// TIA Portal project "Ryan" (V14)

(* hardware
DEVICE "S71500/ET200MP station_1"  S7-1500 station
   slot 0: "Rail_0"  Rack  6ES7 590-1***0-0AA0
   slot 1: "PLC_1"  CPU 1516-3 PN/DP  6ES7 516-3AN01-0AB0  V2.1
      slot 3: "CPU display_1"  6ES7591-1BA00-0AA0
   slot 2: "DI 32x24VDC HF_1"  DI 32x24VDC HF  6ES7 521-1BL00-0AB0  V2.1
   slot 3: "DQ 32x24VDC/0.5A HF_1"  DQ 32x24VDC/0.5A HF  6ES7 522-1BL01-0AB0  V1.0
   slot 4: "AI 8xU/I/RTD/TC ST_1"  AI 8xU/I/RTD/TC ST  6ES7 531-7KF00-0AB0  V2.1
   slot 5: "AQ 4xU/I ST_1"  AQ 4xU/I ST  6ES7 532-5HD00-0AB0  V2.1
DEVICE "PC station"  SIMATIC PC station
   slot 0: "PC station"  Rail  SIMATIC PC-Station  V1.0
      slot 125: "Stationmanager"  Station_Manager  V6.0.4
   slot 1: "IE general_1"  IE General  IE_CP  V8.2.0
   slot 3: "HMI_RT_1"  WinCC RT Advanced  6AV2 104-0xxxx-xxxx  14.0.1.0
      slot 33792: "Host interface"  Host interface
DEVICE "S71500/ET200MP station_2"  S7-1500 station
   slot 0: "Rail_0"  Rack  6ES7 590-1***0-0AA0
   slot 1: "PLC_2"  Unspecific CPU 1500  6ES7 5XX-XXXXX-XXXX  V2.1
*)

// ===== PLC "PLC_1"  CPU 1516-3 PN/DP =====

VAR_GLOBAL   // PLC tag table "Default tag table"
   "p1" AT %M0.0 : Bool;
   "Clock_Byte" AT %MB1687 : Byte;
   "Clock_10Hz" AT %M1687.0 : Bool;
   "Clock_5Hz" AT %M1687.1 : Bool;
   "Clock_2.5Hz" AT %M1687.2 : Bool;
   "Clock_2Hz" AT %M1687.3 : Bool;
   "Clock_1.25Hz" AT %M1687.4 : Bool;
   "Clock_1Hz" AT %M1687.5 : Bool;
   "Clock_0.625Hz" AT %M1687.6 : Bool;
   "Clock_0.5Hz" AT %M1687.7 : Bool;
   "p2" AT %M0.1 : Bool;
   "p3" AT %M0.2 : Bool;
   "p4" AT %M0.3 : Bool;
   "p5" AT %M0.4 : Bool;
   "p6" AT %M0.5 : Bool;
   "p8" AT %M0.7 : Bool;
   "p9" AT %M1.0 : Bool;
   "p11" AT %M1.2 : Bool;
   "p12" AT %M1.3 : Bool;
   "p13" AT %M1.4 : Bool;
   "p15" AT %M1.6 : Bool;
   "p16" AT %M1.7 : Bool;
   "t1" AT %M2.0 : Bool;
   "t2" AT %M2.1 : Bool;
   "t3" AT %M2.2 : Bool;
   "t4" AT %M2.3 : Bool;
   "t5" AT %M2.4 : Bool;
   "t6" AT %M2.5 : Bool;
   "t7" AT %M2.6 : Bool;
   "t8" AT %M2.7 : Bool;
   "t9" AT %M3.0 : Bool;
   "t10" AT %M3.1 : Bool;
   "t12" AT %M3.3 : Bool;
   "t13" AT %M3.4 : Bool;
   "t14" AT %M3.5 : Bool;
   "t16" AT %M3.7 : Bool;
   "t17" AT %M4.0 : Bool;
   "t18" AT %M4.1 : Bool;
   "t20" AT %M4.3 : Bool;
   "t21" AT %M4.4 : Bool;
   "h" AT %IW4 : Int;
   "B" AT %M4.5 : Bool;
   "p17" AT %M4.6 : Bool;
   "p18" AT %M4.7 : Bool;
   "p19" AT %M5.0 : Bool;
   "p20" AT %M5.1 : Bool;
   "p21" AT %M5.2 : Bool;
   "p22" AT %M5.3 : Bool;
   "p23" AT %M5.4 : Bool;
   "t22" AT %M5.5 : Bool;
   "t23" AT %M5.6 : Bool;
   "t24" AT %M5.7 : Bool;
   "t25" AT %M6.0 : Bool;
   "t26" AT %M6.1 : Bool;
   "t27" AT %M6.2 : Bool;
   "NB1" AT %I0.2 : Bool;
   "NB2" AT %I0.5 : Bool;
   "aux1" AT %M6.3 : Bool;
   "aux2" AT %M6.4 : Bool;
   "aux3" AT %M6.5 : Bool;
   "aux4" AT %M6.6 : Bool;
   "aux5" AT %M6.7 : Bool;
   "aux6" AT %M7.0 : Bool;
   "aux7" AT %M7.1 : Bool;
   "aux8" AT %M7.2 : Bool;
   "aux9" AT %M7.3 : Bool;
   "aux10" AT %M7.4 : Bool;
   "aux11" AT %M7.5 : Bool;
   "aux12" AT %M7.6 : Bool;
   "aux13" AT %M7.7 : Bool;
   "aux14" AT %M8.0 : Bool;
   "aux15" AT %M8.1 : Bool;
   "aux16" AT %M8.2 : Bool;
   "aux17" AT %M8.3 : Bool;
   "aux18" AT %M8.4 : Bool;
   "aux19" AT %M8.5 : Bool;
   "aux20" AT %M8.6 : Bool;
   "aux21" AT %M8.7 : Bool;
   "init" AT %M9.0 : Bool;
   "presenceDiscrete" AT %M9.1 : Bool;
   "AcqAddRead" AT %MW0 : Int;
   "AcqAddStart" AT %MW10 : Int;
   "AcqAddStop" AT %MW12 : Int;
   "AcqAddWrite" AT %MW14 : Int;
   "AcqDateObservation" AT %MW16 : Int;
   "AcqError" AT %M18.0 : Bool;
   "AcqNewValues" AT %M24.0 : Bool;
   "AcqRun" AT %M30.0 : Bool;
   "AcqRunPrevious" AT %M30.1 : Bool;
   "step" AT %MW20 : Int;
   "startTable" AT %MW22 : Int;
   "AcqValues" AT %MD26 : DInt;
   "AcqPrevValues" AT %MD32 : DInt;
   "Timer" AT %T0 : Timer;
   "Time" AT %MD36 : Time;
   "InTime" AT %M0.6 : Bool;
   "TimerOutput" AT %M3.2 : Bool;
   "Done_Signal" AT %M40.0 : Bool;
   "Busy" AT %M40.1 : Bool;
   "Error" AT %M40.2 : Bool;
   "Status" AT %MW42 : Word;
   "Done_Write" AT %M44.0 : Bool;
   "Busy_Write" AT %M44.1 : Bool;
   "Error_Write" AT %M44.2 : Bool;
   "Status_Write" AT %MW46 : Word;
   "Done_Open" AT %M48.0 : Bool;
   "Busy_Open" AT %M48.1 : Bool;
   "Error_Open" AT %M48.2 : Bool;
   "Status_Open" AT %MW50 : Word;
   "id" AT %MD52 : DWord;
   "startAcquisition" AT %M3.6 : Bool;
   "stopAcquisition" AT %M4.2 : Bool;
   "DataLogCreated" AT %M9.2 : Bool;
   "aux22" AT %M9.3 : Bool;
   "createDL" AT %M9.4 : Bool;
   "openDL" AT %M9.5 : Bool;
   "writeDL" AT %M9.6 : Bool;
   "DeleteDL" AT %M9.7 : Bool;
   "closeDL" AT %M18.1 : Bool;
   "p24" AT %M18.2 : Bool;
   "p25" AT %M18.3 : Bool;
   "t28" AT %M18.4 : Bool;
   "t29" AT %M18.5 : Bool;
   "aux23" AT %M18.6 : Bool;
   "mag2count" AT %MW56 : Int;
   "aux24" AT %M18.7 : Bool;
   "Tag_1" AT %T30 : Timer;
   "t30" AT %M19.0 : Bool;
   "Tag_2" AT %T31 : Timer;
   "t31" AT %M19.1 : Bool;
   "p26" AT %M19.2 : Bool;
   "p27" AT %M19.3 : Bool;
   "t32" AT %M19.4 : Bool;
   "resetMag2counter" AT %M19.5 : Bool;
   "aux25" AT %M19.6 : Bool;
END_VAR

VAR_GLOBAL   // PLC tag table "IOVEC"
   "o" AT %I1.6 : Bool;
   "m" AT %I1.7 : Bool;
   "s1" AT %I2.2 : Bool;
   "s2" AT %I2.1 : Bool;
   "s3" AT %I2.0 : Bool;
   "r1" AT %I1.5 : Bool;
   "r2" AT %I1.3 : Bool;
   "r3" AT %I1.1 : Bool;
   "f1" AT %I1.4 : Bool;
   "f2" AT %I1.2 : Bool;
   "f3" AT %I1.0 : Bool;
   "rmag1" AT %I0.1 : Bool;
   "rmag2" AT %I0.4 : Bool;
   "fmag1" AT %I0.0 : Bool;
   "fmag2" AT %I0.3 : Bool;
   "Amag1" AT %Q1.0 : Bool;
   "Amag2" AT %Q1.2 : Bool;
   "Retmag1" AT %Q1.1 : Bool;
   "Retmag2" AT %Q1.3 : Bool;
   "C" AT %Q1.4 : Bool;
   "Pus1" AT %Q0.2 : Bool;
   "Pus2" AT %Q0.1 : Bool;
   "Pus3" AT %Q0.0 : Bool;
END_VAR

DATA_BLOCK "Data_block_1"   // DB1
{ S7_Optimized_Access := 'TRUE' }
VERSION : 0.1
   VAR
      "%I0.0" : Bool;
      "%I0.1" : Bool;
      "%I0.2" : Bool;
      "%I0.3" : Bool;
      "%I0.4" : Bool;
      "%I0.5" : Bool;
      "%I1.0" : Bool;
      "%I1.1" : Bool;
      "%I1.2" : Bool;
      "%I1.3" : Bool;
      "%I1.4" : Bool;
      "%I1.5" : Bool;
      "%I1.6" : Bool;
      "%I1.7" : Bool;
      "%I2.0" : Bool;
      "%I2.1" : Bool;
      "%I2.2" : Bool;
      "%IW4" : Int;
      "%Q0.0" : Bool;
      "%Q0.1" : Bool;
      "%Q0.2" : Bool;
      "%Q1.0" : Bool;
      "%Q1.1" : Bool;
      "%Q1.2" : Bool;
      "%Q1.3" : Bool;
      "%Q1.4" : Bool;
   END_VAR
BEGIN
END_DATA_BLOCK

DATA_BLOCK "DataLog_vars"   // DB3
{ S7_Optimized_Access := 'TRUE' }
VERSION : 0.1
   VAR
      "Name" : String := 'iovectors2';
      ID : DWord := 0;
      Headers : String := 'IOvector';
      Data : Struct
         IOvector : DInt;
      END_STRUCT;
   END_VAR
BEGIN
END_DATA_BLOCK

DATA_BLOCK "DataLog_vars2"   // DB7
{ S7_Optimized_Access := 'TRUE' }
VERSION : 0.1
   VAR
      "Name" : String := 'Test201904081147';
      ID : DWord;
      Header : String := 'Time,IOvector';
      Data : Struct
         "Time" : Time;
         IOvector : DInt;
      END_STRUCT;
   END_VAR
BEGIN
END_DATA_BLOCK

DATA_BLOCK "Runtime"   // DB12
{ S7_Optimized_Access := 'TRUE' }
VERSION : 0.1
   VAR
      ob : OB_Any := 123;
      info : Array[0..4] of LTime;
      retval : Array[0..4] of Int;
   END_VAR
BEGIN
END_DATA_BLOCK

DATA_BLOCK "DATALOGDATA"   // DB16
{ S7_Optimized_Access := 'TRUE' }
VERSION : 0.1
   VAR
      IOVECNAMES : Array[0..22] of String;
      IOVEC : Array[0..22] of Bool;
      AcqValues : Array[0..22] of Bool;
      AcqValuesprev : Array[0..22] of Bool;
      Data : Struct
         o : Bool;
         "m" : Bool;
         s1 : Bool;
         s2 : Bool;
         s3 : Bool;
         r1 : Bool;
         r2 : Bool;
         r3 : Bool;
         f1 : Bool;
         f2 : Bool;
         f3 : Bool;
         rmag1 : Bool;
         rmag2 : Bool;
         fmag1 : Bool;
         fmag2 : Bool;
         Amag1 : Bool;
         Amag2 : Bool;
         Retmag1 : Bool;
         Retmag2 : Bool;
         C : Bool;
         Pus1 : Bool;
         Pus2 : Bool;
         Pus3 : Bool;
      END_STRUCT;
      header : String;
      ID : DWord;
   END_VAR
BEGIN
   IOVECNAMES[1] := 'm';
   IOVECNAMES[2] := 's1';
   IOVECNAMES[3] := 's2';
   IOVECNAMES[4] := 's3';
   IOVECNAMES[5] := 'r1';
   IOVECNAMES[6] := 'r2';
   IOVECNAMES[7] := 'r3';
   IOVECNAMES[8] := 'f1';
   IOVECNAMES[9] := 'f2';
   IOVECNAMES[10] := 'f3';
   IOVECNAMES[11] := 'rmag1';
   IOVECNAMES[12] := 'rmag2';
   IOVECNAMES[13] := 'fmag1';
   IOVECNAMES[14] := 'fmag2';
   IOVECNAMES[15] := 'Amag1';
   IOVECNAMES[16] := 'Amag2';
   IOVECNAMES[17] := 'Retmag1';
   IOVECNAMES[18] := 'Retmag2';
   IOVECNAMES[19] := 'C';
   IOVECNAMES[20] := 'Pus1';
   IOVECNAMES[21] := 'Pus2';
   IOVECNAMES[22] := 'Pus3';
   IOVECNAMES[0] := 'o';
END_DATA_BLOCK

DATA_BLOCK "LOGDATA_DB"   // DB17
{ S7_Optimized_Access := 'TRUE' }
VERSION : 0.1
// stored: InstanceOfName LOGDATA
"LOGDATA"
BEGIN
END_DATA_BLOCK

DATA_BLOCK "DATALOG"   // DB18
{ S7_Optimized_Access := 'TRUE' }
VERSION : 0.1
   VAR
      ACQValues : Array[1..23] of Bool;
   END_VAR
BEGIN
END_DATA_BLOCK

// folder: System blocks/Program resources

DATA_BLOCK "IEC_Timer_0_DB"   // DB6
{ S7_Optimized_Access := 'TRUE' }
AUTHOR : Simatic
FAMILY : IEC
NAME : IEC_TMR
VERSION : 1.0
// stored: InstanceOfName IEC_TIMER
"IEC_TIMER"
BEGIN
END_DATA_BLOCK

DATA_BLOCK "IEC_Timer_0_DB_1"   // DB10
{ S7_Optimized_Access := 'TRUE' }
AUTHOR : Simatic
FAMILY : IEC
NAME : IEC_TMR
VERSION : 1.0
// stored: InstanceOfName IEC_TIMER
"IEC_TIMER"
BEGIN
END_DATA_BLOCK

DATA_BLOCK "IEC_Timer_0_DB_2"   // DB11
{ S7_Optimized_Access := 'TRUE' }
AUTHOR : Simatic
FAMILY : IEC
NAME : IEC_TMR
VERSION : 1.0
// stored: InstanceOfName IEC_TIMER
"IEC_TIMER"
BEGIN
END_DATA_BLOCK

DATA_BLOCK "IEC_Timer_0_DB_3"   // DB13
{ S7_Optimized_Access := 'TRUE' }
AUTHOR : Simatic
FAMILY : IEC
NAME : IEC_TMR
VERSION : 1.0
// stored: InstanceOfName IEC_TIMER
"IEC_TIMER"
BEGIN
END_DATA_BLOCK

DATA_BLOCK "IEC_Timer_0_DB_4"   // DB14
{ S7_Optimized_Access := 'TRUE' }
AUTHOR : Simatic
FAMILY : IEC
NAME : IEC_TMR
VERSION : 1.0
// stored: InstanceOfName IEC_TIMER
"IEC_TIMER"
BEGIN
END_DATA_BLOCK

DATA_BLOCK "IEC_Counter_0_DB"   // DB15
{ S7_Optimized_Access := 'TRUE' }
AUTHOR : Simatic
FAMILY : IEC
NAME : CNTR
VERSION : 1.0
// stored: InstanceOfName IEC_COUNTER
"IEC_COUNTER"
BEGIN
END_DATA_BLOCK

// folder: (top level)

ORGANIZATION_BLOCK "Main"   // OB1, LAD, ProgramCycle
TITLE = "Main Program Sweep (Cycle)"
{ S7_Optimized_Access := 'FALSE' }
VERSION : 0.1
   VAR_TEMP
      EV_CLASS : Byte;   // Bits 0-3 = 1:Coming event, Bits 4-7 = 1:Event class 1
      SCAN_1 : Byte;   // 1:Initial call of the OB, 3: Call 2-n of the OB
      PRIORITY : Byte;   // Priority of OB Execution
      OB_NUMBR : Byte;   // OB number
      RESERVED_1 : Byte;   // Reserved for system
      RESERVED_2 : Byte;   // Reserved for system
      PREV_CYCLE : Int;   // Previous program cycle time (milliseconds)
      MIN_CYCLE : Int;   // Minimum program cycle time (milliseconds)
      MAX_CYCLE : Int;   // Maximum program cycle time (milliseconds)
      DATE_TIME : Date_And_Time;   // Date and time OB started
      activateCreate : Bool;
      DataLogAlreadyExists : Bool;
      DeleteDataLog : Bool;
   END_VAR
BEGIN

REGION Network 1
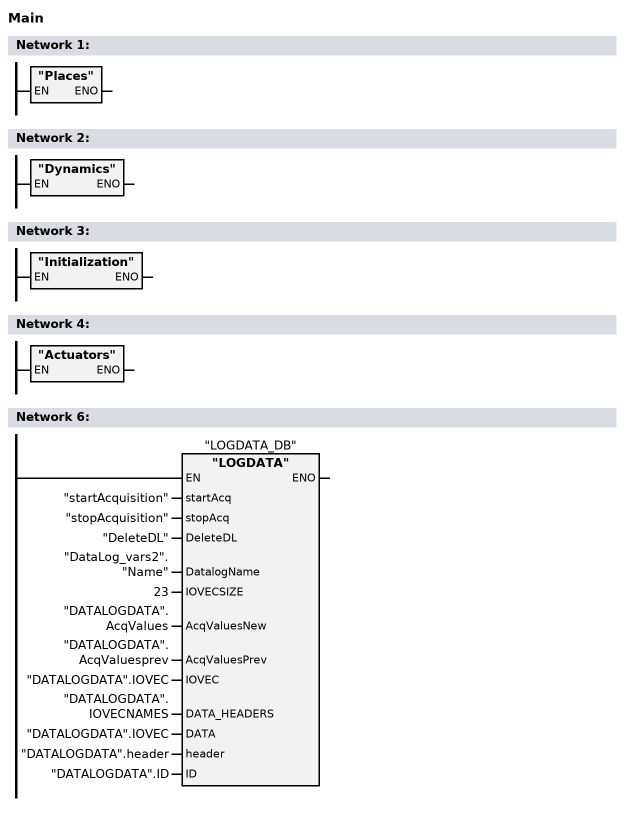
   RUNG wire#powerrail
      "Places"()
   END_RUNG
   // the same network as SCL:
   "Places"();
END_REGION

REGION Network 2
   RUNG wire#powerrail
      "Dynamics"()
   END_RUNG
   // the same network as SCL:
   "Dynamics"();
END_REGION

REGION Network 3
   RUNG wire#powerrail
      "Initialization"()
   END_RUNG
   // the same network as SCL:
   "Initialization"();
END_REGION

REGION Network 4
   RUNG wire#powerrail
      "Actuators"()
   END_RUNG
   // the same network as SCL:
   "Actuators"();
END_REGION

REGION Network 6
   RUNG wire#powerrail
      "LOGDATA_DB"(startAcq := "startAcquisition", stopAcq := "stopAcquisition", DeleteDL := "DeleteDL", DatalogName := "DataLog_vars2"."Name", IOVECSIZE := 23, AcqValuesNew := "DATALOGDATA".AcqValues, AcqValuesPrev := "DATALOGDATA".AcqValuesprev, IOVEC := "DATALOGDATA".IOVEC, DATA_HEADERS := "DATALOGDATA".IOVECNAMES, DATA := "DATALOGDATA".IOVEC, header := "DATALOGDATA".header, ID := "DATALOGDATA".ID)
   END_RUNG
   // the same network as SCL:
   "LOGDATA_DB"(startAcq := "startAcquisition",   // "LOGDATA"
                stopAcq := "stopAcquisition",
                DeleteDL := "DeleteDL",
                DatalogName := "DataLog_vars2"."Name",
                IOVECSIZE := 23,
                AcqValuesNew := "DATALOGDATA".AcqValues,
                AcqValuesPrev := "DATALOGDATA".AcqValuesprev,
                IOVEC := "DATALOGDATA".IOVEC,
                DATA_HEADERS := "DATALOGDATA".IOVECNAMES,
                DATA := "DATALOGDATA".IOVEC,
                header := "DATALOGDATA".header,
                ID := "DATALOGDATA".ID);
END_REGION
END_ORGANIZATION_BLOCK

// folder: LOGGING

FUNCTION_BLOCK "LOGDATA"   // FB1, LAD
{ S7_Optimized_Access := 'TRUE' }
VERSION : 0.1
   VAR_INPUT
      startAcq : Bool;
      stopAcq : Bool;
      DeleteDL : Bool;
      DatalogName : String;
      IOVECSIZE : UDInt;
   END_VAR
   VAR_IN_OUT
      AcqValuesNew : Array[*] of Bool;
      AcqValuesPrev : Array[*] of Bool;
      IOVEC : Array[*] of Bool;
      DATA_HEADERS : Array[*] of String;
      DATA : Variant;
      header : String;
      ID : DWord;
   END_VAR
   VAR_TEMP
      DeleteDatalog : Bool;
      moveBlkVariantRetVal : Int;
      i : Int;
      dataheaderslowerbound : DInt;
      dataheadersupperbound : DInt;
   END_VAR
   VAR_TEMP   // added for the SCL form of the ladder/FBD networks
      _w1 : Bool;
      _w2 : Bool;
   END_VAR
BEGIN

REGION Network 1 (SCL): Name header
       #header := '';
   #dataheaderslowerbound := LOWER_BOUND(ARR := #DATA_HEADERS, DIM := 1);
   #dataheadersupperbound := UPPER_BOUND(ARR := #DATA_HEADERS, DIM := 1);

   FOR #i := #dataheaderslowerbound TO #dataheadersupperbound-1 DO
       // Statement section FOR

       #header := CONCAT(IN1 := #header, IN2 := #DATA_HEADERS[#i]);
       #header := CONCAT(IN1 := #header, IN2 := ',');
   END_FOR;
   #header := CONCAT(IN1 := #header, IN2 := #DATA_HEADERS[#dataheadersupperbound]);
END_REGION

REGION Network 2: Start or stop acquisition
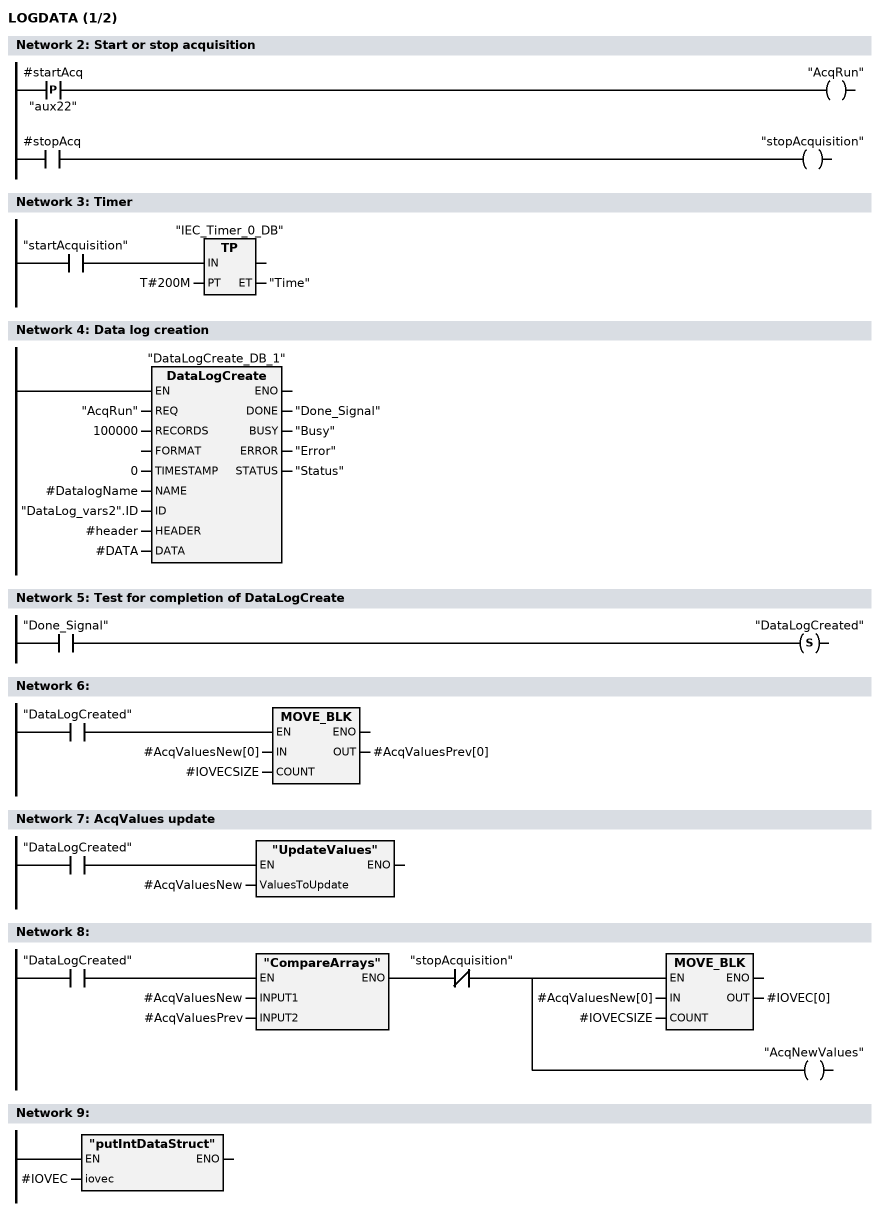
   RUNG wire#powerrail
      P_Contact(operand := #startAcq, bit := "aux22")
      Coil( "AcqRun" )
   END_RUNG
   RUNG wire#powerrail
      Contact( #stopAcq )
      Coil( "stopAcquisition" )
   END_RUNG
   // the same network as SCL:
   #_w1 := #startAcq AND NOT "aux22";   // rising edge of #startAcq
   "aux22" := #startAcq;
   "AcqRun" := #_w1;
   "stopAcquisition" := #stopAcq;
END_REGION

REGION Network 3: Timer
   "IEC_Timer_0_DB".TP(IN := "startAcquisition", PT := T#200M, ET => "Time");
END_REGION

REGION Network 4: Data log creation
   "DataLogCreate_DB_1"(REQ := "AcqRun",   // DataLogCreate
                        RECORDS := 100000,
                        TIMESTAMP := 0,
                        "NAME" := #DatalogName,
                        ID := "DataLog_vars2".ID,
                        HEADER := #header,
                        DATA := #DATA,
                        DONE => "Done_Signal",
                        BUSY => "Busy",
                        ERROR => "Error",
                        STATUS => "Status");
END_REGION

REGION Network 5: Test for completion of DataLogCreate
   RUNG wire#powerrail
      Contact( "Done_Signal" )
      S_Coil( "DataLogCreated" )
   END_RUNG
   // the same network as SCL:
   IF "Done_Signal" THEN "DataLogCreated" := TRUE; END_IF;
END_REGION

REGION Network 6
   IF "DataLogCreated" THEN
       MOVE_BLK(IN := #AcqValuesNew[0], COUNT := #IOVECSIZE, OUT => #AcqValuesPrev[0]);
   END_IF;
END_REGION

REGION Network 7: AcqValues update
   RUNG wire#powerrail
      Contact( "DataLogCreated" )
      "UpdateValues"(ValuesToUpdate := #AcqValuesNew)
   END_RUNG
   // the same network as SCL:
   IF "DataLogCreated" THEN "UpdateValues"(ValuesToUpdate := #AcqValuesNew); END_IF;
END_REGION

REGION Network 8
   "CompareArrays"(EN := "DataLogCreated", INPUT1 := #AcqValuesNew, INPUT2 := #AcqValuesPrev, ENO => #_w1);
   #_w2 := #_w1 AND NOT "stopAcquisition";
   IF #_w2 THEN MOVE_BLK(IN := #AcqValuesNew[0], COUNT := #IOVECSIZE, OUT => #IOVEC[0]); END_IF;
   "AcqNewValues" := #_w2;
END_REGION

REGION Network 9
   RUNG wire#powerrail
      "putIntDataStruct"(iovec := #IOVEC)
   END_RUNG
   // the same network as SCL:
   "putIntDataStruct"(iovec := #IOVEC);
END_REGION

REGION Network 10: Write to data log
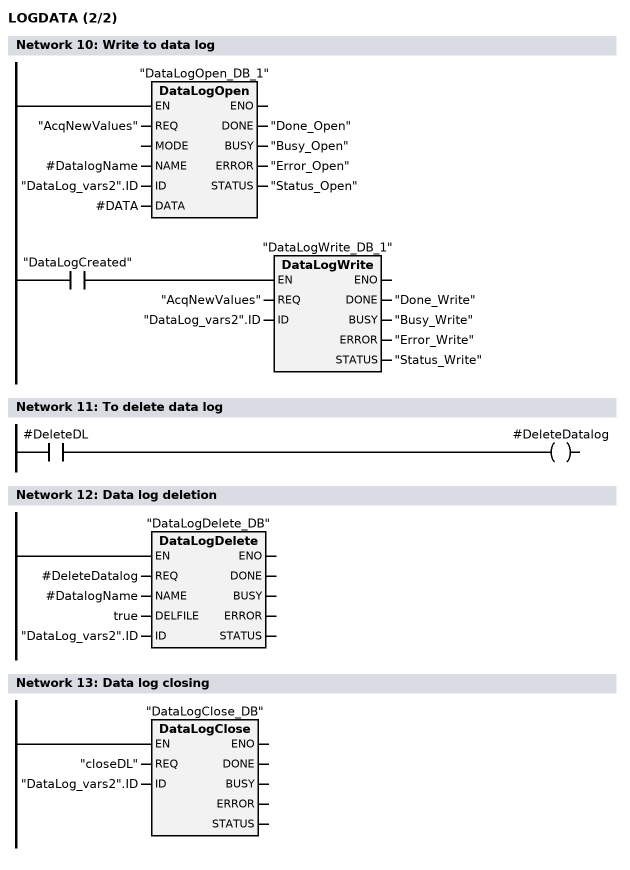
   "DataLogOpen_DB_1"(REQ := "AcqNewValues",   // DataLogOpen
                      "NAME" := #DatalogName,
                      ID := "DataLog_vars2".ID,
                      Data := #DATA,
                      DONE => "Done_Open",
                      BUSY => "Busy_Open",
                      ERROR => "Error_Open",
                      STATUS => "Status_Open");
   IF "DataLogCreated" THEN
       "DataLogWrite_DB_1"(REQ := "AcqNewValues",   // DataLogWrite
                           ID := "DataLog_vars2".ID,
                           DONE => "Done_Write",
                           BUSY => "Busy_Write",
                           ERROR => "Error_Write",
                           STATUS => "Status_Write");
   END_IF;
END_REGION

REGION Network 11: To delete data log
   RUNG wire#powerrail
      Contact( #DeleteDL )
      Coil( #DeleteDatalog )
   END_RUNG
   // the same network as SCL:
   #DeleteDatalog := #DeleteDL;
END_REGION

REGION Network 12: Data log deletion
   "DataLogDelete_DB"(REQ := #DeleteDatalog, "NAME" := #DatalogName, DelFile := true, ID := "DataLog_vars2".ID);   // DataLogDelete
END_REGION

REGION Network 13: Data log closing
   "DataLogClose_DB"(REQ := "closeDL", ID := "DataLog_vars2".ID);   // DataLogClose
END_REGION
END_FUNCTION_BLOCK

FUNCTION "DataLogging" : Void   // FC5, LAD
{ S7_Optimized_Access := 'TRUE' }
VERSION : 0.1
   VAR_INPUT
      startAcq : Bool;
      stopAcq : Bool;
      DeleteDL : Bool;
      DatalogName : String;
   END_VAR
   VAR_TEMP
      DeleteDatalog : Bool;
   END_VAR
   VAR_TEMP   // added for the SCL form of the ladder/FBD networks
      _w1 : Bool;
   END_VAR
BEGIN

REGION Network 1: Start or stop acquisition
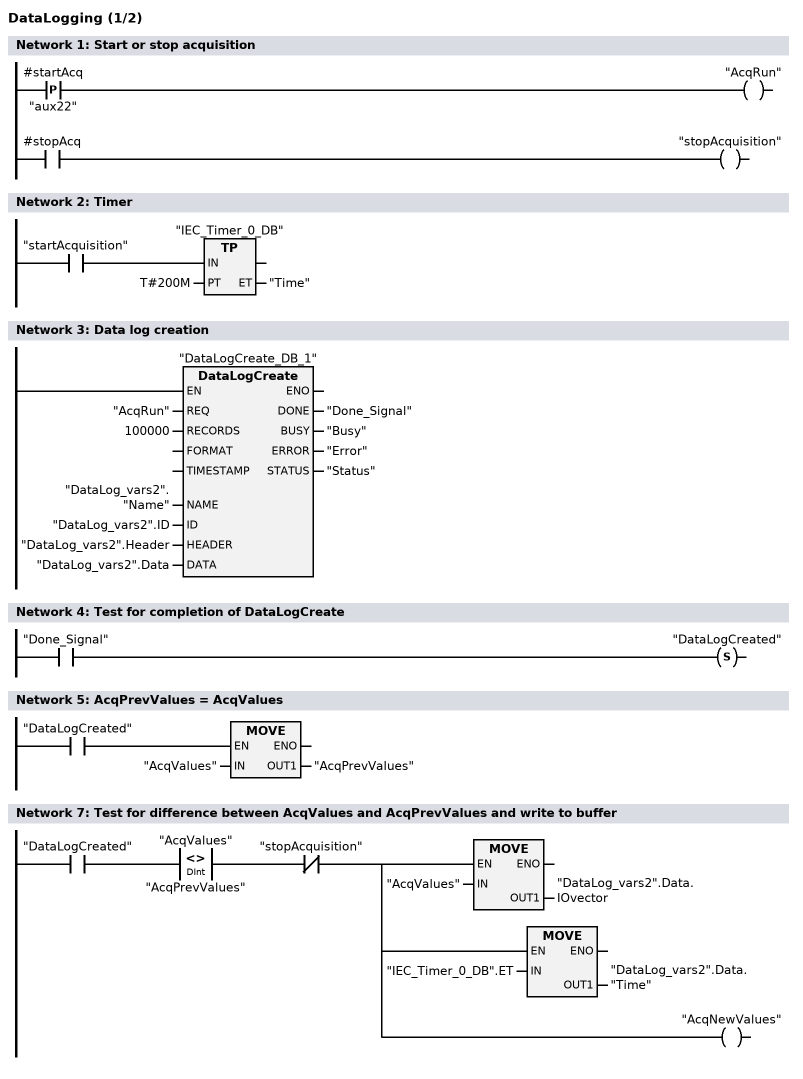
   RUNG wire#powerrail
      P_Contact(operand := #startAcq, bit := "aux22")
      Coil( "AcqRun" )
   END_RUNG
   RUNG wire#powerrail
      Contact( #stopAcq )
      Coil( "stopAcquisition" )
   END_RUNG
   // the same network as SCL:
   #_w1 := #startAcq AND NOT "aux22";   // rising edge of #startAcq
   "aux22" := #startAcq;
   "AcqRun" := #_w1;
   "stopAcquisition" := #stopAcq;
END_REGION

REGION Network 2: Timer
   "IEC_Timer_0_DB".TP(IN := "startAcquisition", PT := T#200M, ET => "Time");
END_REGION

REGION Network 3: Data log creation
   "DataLogCreate_DB_1"(REQ := "AcqRun",   // DataLogCreate
                        RECORDS := 100000,
                        "NAME" := "DataLog_vars2"."Name",
                        ID := "DataLog_vars2".ID,
                        HEADER := "DataLog_vars2".Header,
                        DATA := "DataLog_vars2".Data,
                        DONE => "Done_Signal",
                        BUSY => "Busy",
                        ERROR => "Error",
                        STATUS => "Status");
END_REGION

REGION Network 4: Test for completion of DataLogCreate
   RUNG wire#powerrail
      Contact( "Done_Signal" )
      S_Coil( "DataLogCreated" )
   END_RUNG
   // the same network as SCL:
   IF "Done_Signal" THEN "DataLogCreated" := TRUE; END_IF;
END_REGION

REGION Network 5: AcqPrevValues = AcqValues
   RUNG wire#powerrail
      Contact( "DataLogCreated" )
      Move(in := "AcqValues", out1 => "AcqPrevValues")
   END_RUNG
   // the same network as SCL:
   IF "DataLogCreated" THEN "AcqPrevValues" := "AcqValues"; END_IF;
END_REGION

REGION Network 6 (SCL): AcqValues update
   IF "DataLogCreated" THEN
       "AcqValues".%X0 := "fmag1";
       "AcqValues".%X1 := "rmag1";
       "AcqValues".%X2 := "fmag2";
       "AcqValues".%X3 := "rmag2";
       "AcqValues".%X4 := "f3";
       "AcqValues".%X5 := "r3";
       "AcqValues".%X6 := "f2";
       "AcqValues".%X7 := "r2";
       "AcqValues".%X8 := "f1";
       "AcqValues".%X9 := "r1";
       "AcqValues".%X10 := "o";
       "AcqValues".%X11 := "m";
       "AcqValues".%X12 := "s3";
       "AcqValues".%X13 := "s2";
       "AcqValues".%X14 := "s1";
       "AcqValues".%X15 := "Pus3";
       "AcqValues".%X16 := "Pus2";
       "AcqValues".%X17 := "Pus1";
       "AcqValues".%X18 := "Amag1";
       "AcqValues".%X19 := "Retmag1";
       "AcqValues".%X20 := "Amag2";
       "AcqValues".%X21 := "Retmag2";
       "AcqValues".%X22 := "C";
   END_IF;
END_REGION

REGION Network 7: Test for difference between AcqValues and AcqPrevValues and write to buffer
   RUNG wire#powerrail
      Contact( "DataLogCreated" )
      { S7_Templates := "SrcType := DInt" } NE_Contact(in1 := "AcqValues", in2 := "AcqPrevValues")
      I_Contact( "stopAcquisition" )
      wire#w1
      Move(in := "AcqValues", out1 => "DataLog_vars2".Data.IOvector)
   END_RUNG
   RUNG wire#w1
      Move(in := "IEC_Timer_0_DB".ET, out1 => "DataLog_vars2".Data."Time")
   END_RUNG
   RUNG wire#w1
      Coil( "AcqNewValues" )
   END_RUNG
   // the same network as SCL:
   #_w1 := "DataLogCreated" AND ("AcqValues" <> "AcqPrevValues") AND NOT "stopAcquisition";
   IF #_w1 THEN
       "DataLog_vars2".Data.IOvector := "AcqValues";
       "DataLog_vars2".Data."Time" := "IEC_Timer_0_DB".ET;
   END_IF;
   "AcqNewValues" := #_w1;
END_REGION

REGION Network 8: Write to data log
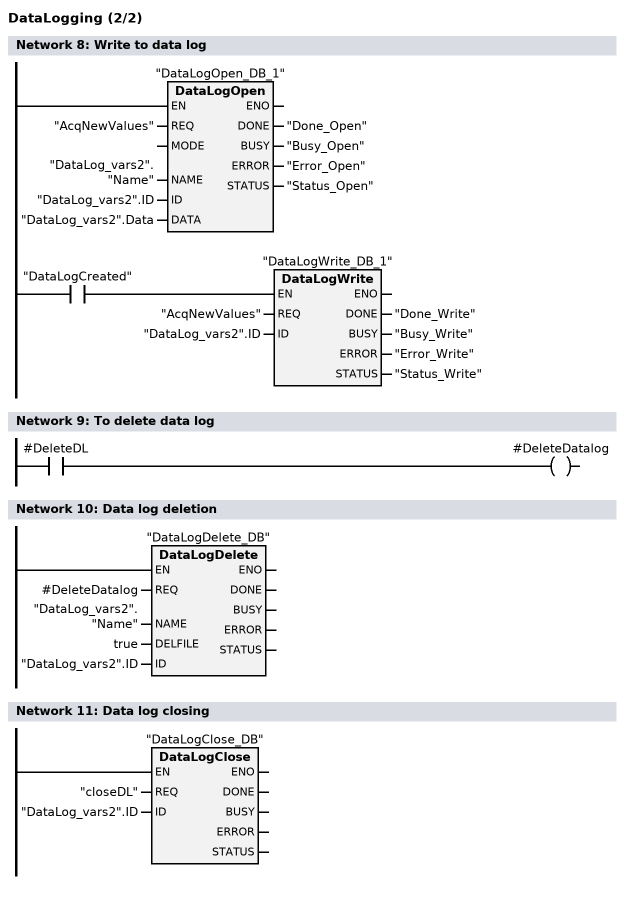
   "DataLogOpen_DB_1"(REQ := "AcqNewValues",   // DataLogOpen
                      "NAME" := "DataLog_vars2"."Name",
                      ID := "DataLog_vars2".ID,
                      Data := "DataLog_vars2".Data,
                      DONE => "Done_Open",
                      BUSY => "Busy_Open",
                      ERROR => "Error_Open",
                      STATUS => "Status_Open");
   IF "DataLogCreated" THEN
       "DataLogWrite_DB_1"(REQ := "AcqNewValues",   // DataLogWrite
                           ID := "DataLog_vars2".ID,
                           DONE => "Done_Write",
                           BUSY => "Busy_Write",
                           ERROR => "Error_Write",
                           STATUS => "Status_Write");
   END_IF;
END_REGION

REGION Network 9: To delete data log
   RUNG wire#powerrail
      Contact( #DeleteDL )
      Coil( #DeleteDatalog )
   END_RUNG
   // the same network as SCL:
   #DeleteDatalog := #DeleteDL;
END_REGION

REGION Network 10: Data log deletion
   "DataLogDelete_DB"(REQ := #DeleteDatalog,   // DataLogDelete
                      "NAME" := "DataLog_vars2"."Name",
                      DelFile := true,
                      ID := "DataLog_vars2".ID);
END_REGION

REGION Network 11: Data log closing
   "DataLogClose_DB"(REQ := "closeDL", ID := "DataLog_vars2".ID);   // DataLogClose
END_REGION

REGION Network 12 (SCL)
   "Runtime".ob := "OB_Main";

   "Runtime".retval[1] := RT_INFO(MODE := 1,
                                  OB := "Runtime".ob,
                                  INFO := "Runtime".info[1]);

   "Runtime".retval[2] := RT_INFO(MODE := 2,
                                  OB := "Runtime".ob,
                                  INFO := "Runtime".info[2]);

   "Runtime".retval[3] := RT_INFO(MODE := 3,
                                  OB := "Runtime".ob,
                                  INFO := "Runtime".info[3]);

   "Runtime".retval[4] := RT_INFO(MODE := 25,
                                  OB := "Runtime".ob,
                                  INFO := "Runtime".info[4]);
END_REGION
END_FUNCTION

FUNCTION "UpdateValues" : Void   // FC6, LAD
{ S7_Optimized_Access := 'TRUE' }
VERSION : 0.1
   VAR_IN_OUT
      ValuesToUpdate : Array[*] of Bool;
   END_VAR
BEGIN

REGION Network 1 (SCL)
   #ValuesToUpdate[0] := "o";
   #ValuesToUpdate[1] := "m";
   #ValuesToUpdate[2] := "s1";
   #ValuesToUpdate[3] := "s2";
   #ValuesToUpdate[4] := "s3";
   #ValuesToUpdate[5] := "r1";
   #ValuesToUpdate[6] := "r2";
   #ValuesToUpdate[7] := "r3";
   #ValuesToUpdate[8] := "f1";
   #ValuesToUpdate[9] := "f2";
   #ValuesToUpdate[10] := "f3";
   #ValuesToUpdate[11] := "rmag1";
   #ValuesToUpdate[12] := "rmag2";
   #ValuesToUpdate[13] := "fmag1";
   #ValuesToUpdate[14] := "fmag2";
   #ValuesToUpdate[15] := "Amag1";
   #ValuesToUpdate[16] := "Amag2";
   #ValuesToUpdate[17] := "Retmag1";
   #ValuesToUpdate[18] := "Retmag2";
   #ValuesToUpdate[19] := "C";
   #ValuesToUpdate[20] := "Pus1";
   #ValuesToUpdate[21] := "Pus2";
   #ValuesToUpdate[22] := "Pus3";
END_REGION
END_FUNCTION

FUNCTION "putIntDataStruct" : Void   // FC8, LAD
{ S7_Optimized_Access := 'TRUE' }
VERSION : 0.1
   VAR_IN_OUT
      iovec : Array[*] of Bool;
   END_VAR
BEGIN

REGION Network 1 (SCL)
   "DATALOGDATA".Data.o := #iovec[0];
   "DATALOGDATA".Data."m" := #iovec[1];
   "DATALOGDATA".Data.s1 := #iovec[2];
   "DATALOGDATA".Data.s2 := #iovec[3];
   "DATALOGDATA".Data.s3 := #iovec[4];
   "DATALOGDATA".Data.r1 := #iovec[5];
   "DATALOGDATA".Data.r2 := #iovec[6];
   "DATALOGDATA".Data.r3 := #iovec[7];
   "DATALOGDATA".Data.f1 := #iovec[8];
   "DATALOGDATA".Data.f2 := #iovec[9];
   "DATALOGDATA".Data.f3 := #iovec[10];
   "DATALOGDATA".Data.rmag1 := #iovec[11];
   "DATALOGDATA".Data.rmag2 := #iovec[12];
   "DATALOGDATA".Data.fmag1 := #iovec[13];
   "DATALOGDATA".Data.fmag2 := #iovec[14];
   "DATALOGDATA".Data.Amag1 := #iovec[15];
   "DATALOGDATA".Data.Amag2 := #iovec[16];
   "DATALOGDATA".Data.Retmag1 := #iovec[17];
   "DATALOGDATA".Data.Retmag2 := #iovec[18];
   "DATALOGDATA".Data.C := #iovec[19];
   "DATALOGDATA".Data.Pus1 := #iovec[20];
   "DATALOGDATA".Data.Pus2 := #iovec[21];
   "DATALOGDATA".Data.Pus3 := #iovec[22];
END_REGION
END_FUNCTION

// folder: LOGGING/utils

FUNCTION "CompareArrays" : Void   // FC7, LAD
{ S7_Optimized_Access := 'TRUE' }
VERSION : 0.1
   VAR_INPUT
      INPUT1 : Array[*] of Bool;
      INPUT2 : Array[*] of Bool;
   END_VAR
   VAR_TEMP
      out : Bool;
      i : Int;
      dataheaderslowerbound : DInt;
      dataheadersupperbound : DInt;
   END_VAR
BEGIN

REGION Network 1 (SCL)
   #out := TRUE;

   #dataheaderslowerbound := LOWER_BOUND(ARR := #INPUT1, DIM := 1);
   #dataheadersupperbound := UPPER_BOUND(ARR := #INPUT1, DIM := 1);

   FOR #i := #dataheaderslowerbound TO #dataheadersupperbound DO
       // Statement section FOR
       #out := #out AND (#INPUT1[#i] = #INPUT2[#i]);

   END_FOR;

   ENO := NOT #out;
END_REGION
END_FUNCTION

// folder: PetriNet

FUNCTION "Places" : Void   // FC1, LAD
{ S7_Optimized_Access := 'TRUE' }
VERSION : 0.1
   VAR_TEMP   // added for the SCL form of the ladder/FBD networks
      _w1 : Bool;
      _w2 : Bool;
      _w3 : Bool;
      _w4 : Bool;
      _w5 : Bool;
      _w6 : Bool;
      _w7 : Bool;
      _w8 : Bool;
      _w9 : Bool;
      _w10 : Bool;
      _w11 : Bool;
      _w12 : Bool;
      _w13 : Bool;
      _w14 : Bool;
      _w15 : Bool;
      _w16 : Bool;
      _w17 : Bool;
      _w18 : Bool;
   END_VAR
BEGIN

REGION Network 1
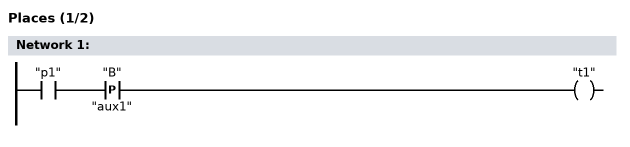
   RUNG wire#powerrail
      Contact( "p1" )
      P_Contact(operand := "B", bit := "aux1")
      Coil( "t1" )
   END_RUNG
   // the same network as SCL:
   #_w1 := "p1" AND "B" AND NOT "aux1";   // rising edge of "B"
   "aux1" := "B";
   "t1" := #_w1;
END_REGION

REGION Network 2: Places
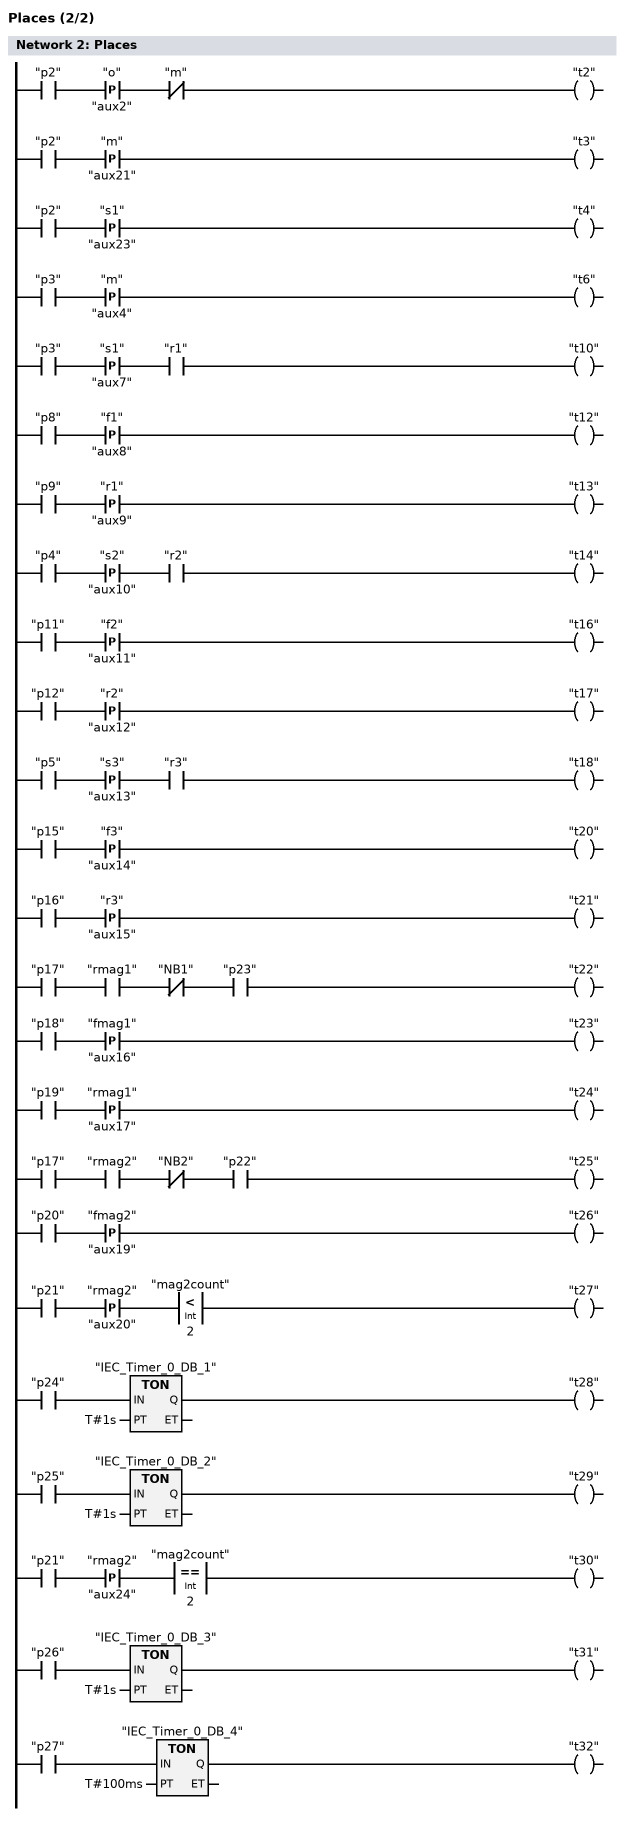
   #_w1 := "p2" AND "o" AND NOT "aux2";   // rising edge of "o"
   "aux2" := "o";
   "t2" := #_w1 AND NOT "m";
   #_w2 := "p2" AND "m" AND NOT "aux21";   // rising edge of "m"
   "aux21" := "m";
   "t3" := #_w2;
   #_w3 := "p2" AND "s1" AND NOT "aux23";   // rising edge of "s1"
   "aux23" := "s1";
   "t4" := #_w3;
   #_w4 := "p3" AND "m" AND NOT "aux4";   // rising edge of "m"
   "aux4" := "m";
   "t6" := #_w4;
   #_w5 := "p3" AND "s1" AND NOT "aux7";   // rising edge of "s1"
   "aux7" := "s1";
   "t10" := #_w5 AND "r1";
   #_w6 := "p8" AND "f1" AND NOT "aux8";   // rising edge of "f1"
   "aux8" := "f1";
   "t12" := #_w6;
   #_w7 := "p9" AND "r1" AND NOT "aux9";   // rising edge of "r1"
   "aux9" := "r1";
   "t13" := #_w7;
   #_w8 := "p4" AND "s2" AND NOT "aux10";   // rising edge of "s2"
   "aux10" := "s2";
   "t14" := #_w8 AND "r2";
   #_w9 := "p11" AND "f2" AND NOT "aux11";   // rising edge of "f2"
   "aux11" := "f2";
   "t16" := #_w9;
   #_w10 := "p12" AND "r2" AND NOT "aux12";   // rising edge of "r2"
   "aux12" := "r2";
   "t17" := #_w10;
   #_w11 := "p5" AND "s3" AND NOT "aux13";   // rising edge of "s3"
   "aux13" := "s3";
   "t18" := #_w11 AND "r3";
   #_w12 := "p15" AND "f3" AND NOT "aux14";   // rising edge of "f3"
   "aux14" := "f3";
   "t20" := #_w12;
   #_w13 := "p16" AND "r3" AND NOT "aux15";   // rising edge of "r3"
   "aux15" := "r3";
   "t21" := #_w13;
   "t22" := "p17" AND "rmag1" AND NOT "NB1" AND "p23";
   #_w14 := "p18" AND "fmag1" AND NOT "aux16";   // rising edge of "fmag1"
   "aux16" := "fmag1";
   "t23" := #_w14;
   #_w15 := "p19" AND "rmag1" AND NOT "aux17";   // rising edge of "rmag1"
   "aux17" := "rmag1";
   "t24" := #_w15;
   "t25" := "p17" AND "rmag2" AND NOT "NB2" AND "p22";
   #_w16 := "p20" AND "fmag2" AND NOT "aux19";   // rising edge of "fmag2"
   "aux19" := "fmag2";
   "t26" := #_w16;
   #_w17 := "p21" AND "rmag2" AND NOT "aux20";   // rising edge of "rmag2"
   "aux20" := "rmag2";
   "t27" := #_w17 AND ("mag2count" < 2);
   "IEC_Timer_0_DB_1".TON(IN := "p24", PT := T#1s);
   "t28" := "IEC_Timer_0_DB_1".Q;
   "IEC_Timer_0_DB_2".TON(IN := "p25", PT := T#1s);
   "t29" := "IEC_Timer_0_DB_2".Q;
   #_w18 := "p21" AND "rmag2" AND NOT "aux24";   // rising edge of "rmag2"
   "aux24" := "rmag2";
   "t30" := #_w18 AND ("mag2count" = 2);
   "IEC_Timer_0_DB_3".TON(IN := "p26", PT := T#1s);
   "t31" := "IEC_Timer_0_DB_3".Q;
   "IEC_Timer_0_DB_4".TON(IN := "p27", PT := T#100ms);
   "t32" := "IEC_Timer_0_DB_4".Q;
END_REGION
END_FUNCTION

FUNCTION "Dynamics" : Void   // FC2, LAD
{ S7_Optimized_Access := 'TRUE' }
VERSION : 0.1
BEGIN

REGION Network 1: Dynamics
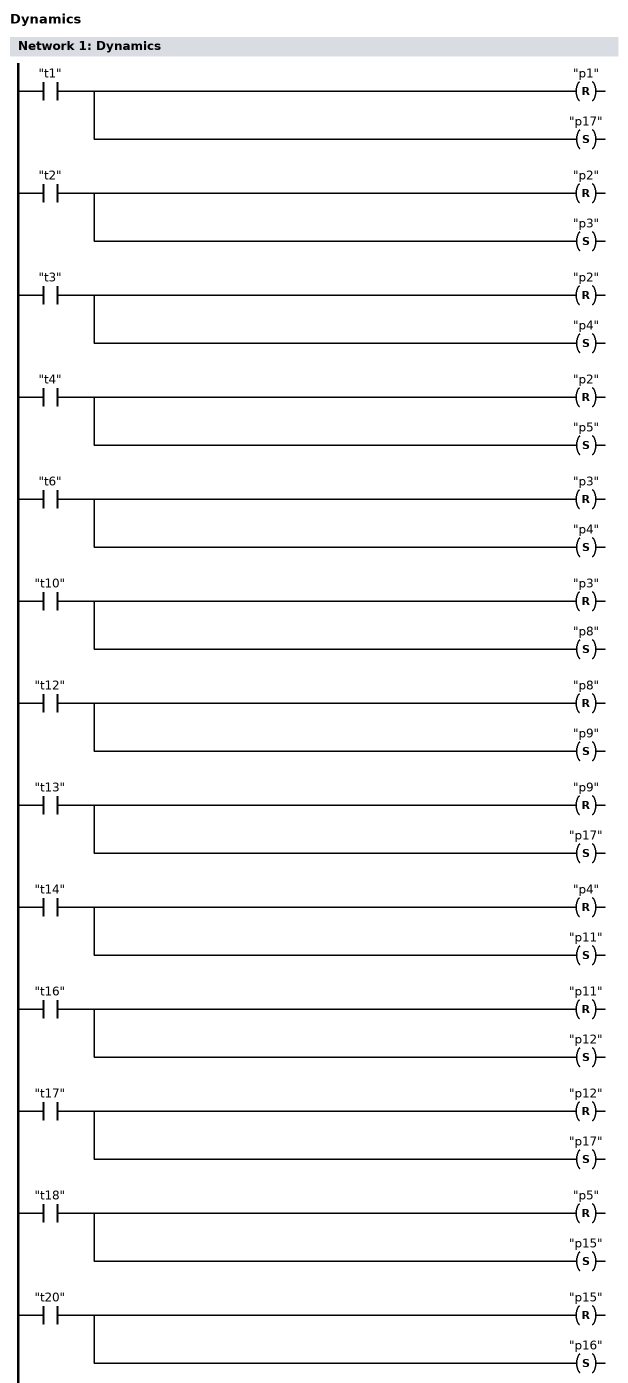
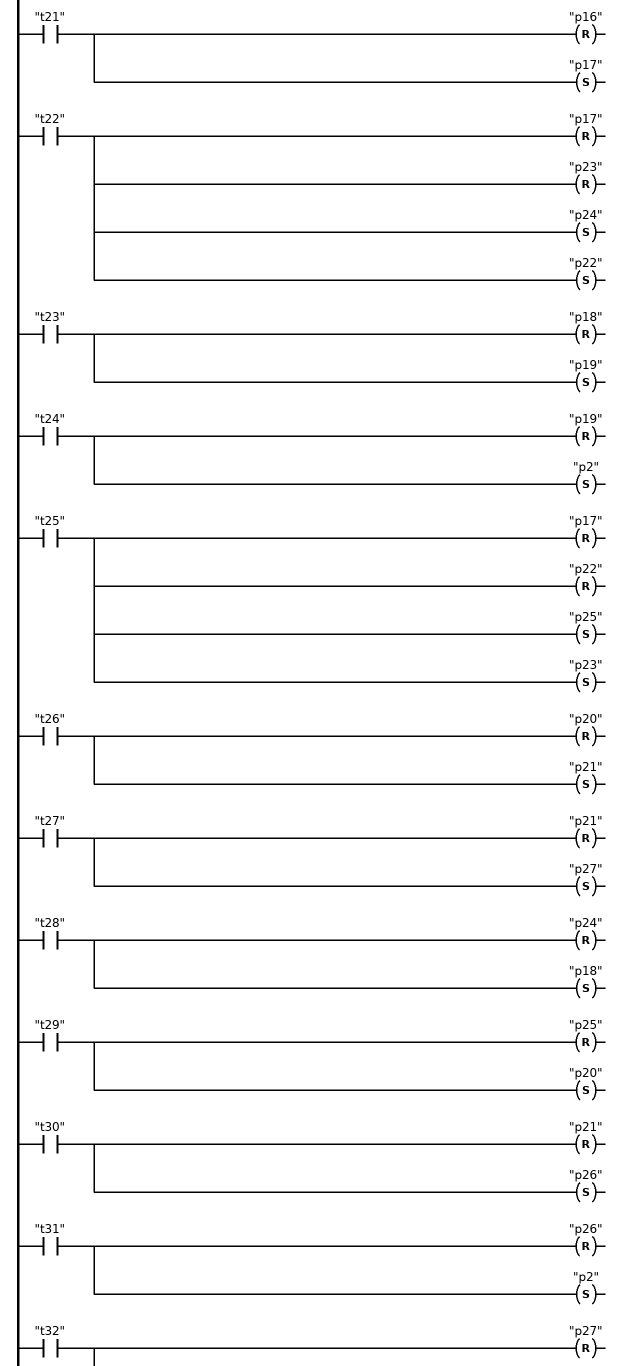
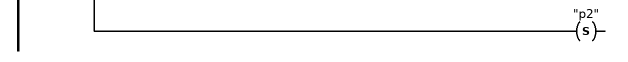
   RUNG wire#powerrail
      Contact( "t1" )
      wire#w1
      R_Coil( "p1" )
   END_RUNG
   RUNG wire#w1
      S_Coil( "p17" )
   END_RUNG
   RUNG wire#powerrail
      Contact( "t2" )
      wire#w2
      R_Coil( "p2" )
   END_RUNG
   RUNG wire#w2
      S_Coil( "p3" )
   END_RUNG
   RUNG wire#powerrail
      Contact( "t3" )
      wire#w3
      R_Coil( "p2" )
   END_RUNG
   RUNG wire#w3
      S_Coil( "p4" )
   END_RUNG
   RUNG wire#powerrail
      Contact( "t4" )
      wire#w4
      R_Coil( "p2" )
   END_RUNG
   RUNG wire#w4
      S_Coil( "p5" )
   END_RUNG
   RUNG wire#powerrail
      Contact( "t6" )
      wire#w5
      R_Coil( "p3" )
   END_RUNG
   RUNG wire#w5
      S_Coil( "p4" )
   END_RUNG
   RUNG wire#powerrail
      Contact( "t10" )
      wire#w6
      R_Coil( "p3" )
   END_RUNG
   RUNG wire#w6
      S_Coil( "p8" )
   END_RUNG
   RUNG wire#powerrail
      Contact( "t12" )
      wire#w7
      R_Coil( "p8" )
   END_RUNG
   RUNG wire#w7
      S_Coil( "p9" )
   END_RUNG
   RUNG wire#powerrail
      Contact( "t13" )
      wire#w8
      R_Coil( "p9" )
   END_RUNG
   RUNG wire#w8
      S_Coil( "p17" )
   END_RUNG
   RUNG wire#powerrail
      Contact( "t14" )
      wire#w9
      R_Coil( "p4" )
   END_RUNG
   RUNG wire#w9
      S_Coil( "p11" )
   END_RUNG
   RUNG wire#powerrail
      Contact( "t16" )
      wire#w10
      R_Coil( "p11" )
   END_RUNG
   RUNG wire#w10
      S_Coil( "p12" )
   END_RUNG
   RUNG wire#powerrail
      Contact( "t17" )
      wire#w11
      R_Coil( "p12" )
   END_RUNG
   RUNG wire#w11
      S_Coil( "p17" )
   END_RUNG
   RUNG wire#powerrail
      Contact( "t18" )
      wire#w12
      R_Coil( "p5" )
   END_RUNG
   RUNG wire#w12
      S_Coil( "p15" )
   END_RUNG
   RUNG wire#powerrail
      Contact( "t20" )
      wire#w13
      R_Coil( "p15" )
   END_RUNG
   RUNG wire#w13
      S_Coil( "p16" )
   END_RUNG
   RUNG wire#powerrail
      Contact( "t21" )
      wire#w14
      R_Coil( "p16" )
   END_RUNG
   RUNG wire#w14
      S_Coil( "p17" )
   END_RUNG
   RUNG wire#powerrail
      Contact( "t22" )
      wire#w15
      R_Coil( "p17" )
   END_RUNG
   RUNG wire#w15
      R_Coil( "p23" )
   END_RUNG
   RUNG wire#w15
      S_Coil( "p24" )
   END_RUNG
   RUNG wire#w15
      S_Coil( "p22" )
   END_RUNG
   RUNG wire#powerrail
      Contact( "t23" )
      wire#w16
      R_Coil( "p18" )
   END_RUNG
   RUNG wire#w16
      S_Coil( "p19" )
   END_RUNG
   RUNG wire#powerrail
      Contact( "t24" )
      wire#w17
      R_Coil( "p19" )
   END_RUNG
   RUNG wire#w17
      S_Coil( "p2" )
   END_RUNG
   RUNG wire#powerrail
      Contact( "t25" )
      wire#w18
      R_Coil( "p17" )
   END_RUNG
   RUNG wire#w18
      R_Coil( "p22" )
   END_RUNG
   RUNG wire#w18
      S_Coil( "p25" )
   END_RUNG
   RUNG wire#w18
      S_Coil( "p23" )
   END_RUNG
   RUNG wire#powerrail
      Contact( "t26" )
      wire#w19
      R_Coil( "p20" )
   END_RUNG
   RUNG wire#w19
      S_Coil( "p21" )
   END_RUNG
   RUNG wire#powerrail
      Contact( "t27" )
      wire#w20
      R_Coil( "p21" )
   END_RUNG
   RUNG wire#w20
      S_Coil( "p27" )
   END_RUNG
   RUNG wire#powerrail
      Contact( "t28" )
      wire#w21
      R_Coil( "p24" )
   END_RUNG
   RUNG wire#w21
      S_Coil( "p18" )
   END_RUNG
   RUNG wire#powerrail
      Contact( "t29" )
      wire#w22
      R_Coil( "p25" )
   END_RUNG
   RUNG wire#w22
      S_Coil( "p20" )
   END_RUNG
   RUNG wire#powerrail
      Contact( "t30" )
      wire#w23
      R_Coil( "p21" )
   END_RUNG
   RUNG wire#w23
      S_Coil( "p26" )
   END_RUNG
   RUNG wire#powerrail
      Contact( "t31" )
      wire#w24
      R_Coil( "p26" )
   END_RUNG
   RUNG wire#w24
      S_Coil( "p2" )
   END_RUNG
   RUNG wire#powerrail
      Contact( "t32" )
      wire#w25
      R_Coil( "p27" )
   END_RUNG
   RUNG wire#w25
      S_Coil( "p2" )
   END_RUNG
   // the same network as SCL:
   IF "t1" THEN
       "p1" := FALSE;
       "p17" := TRUE;
   END_IF;
   IF "t2" THEN
       "p2" := FALSE;
       "p3" := TRUE;
   END_IF;
   IF "t3" THEN
       "p2" := FALSE;
       "p4" := TRUE;
   END_IF;
   IF "t4" THEN
       "p2" := FALSE;
       "p5" := TRUE;
   END_IF;
   IF "t6" THEN
       "p3" := FALSE;
       "p4" := TRUE;
   END_IF;
   IF "t10" THEN
       "p3" := FALSE;
       "p8" := TRUE;
   END_IF;
   IF "t12" THEN
       "p8" := FALSE;
       "p9" := TRUE;
   END_IF;
   IF "t13" THEN
       "p9" := FALSE;
       "p17" := TRUE;
   END_IF;
   IF "t14" THEN
       "p4" := FALSE;
       "p11" := TRUE;
   END_IF;
   IF "t16" THEN
       "p11" := FALSE;
       "p12" := TRUE;
   END_IF;
   IF "t17" THEN
       "p12" := FALSE;
       "p17" := TRUE;
   END_IF;
   IF "t18" THEN
       "p5" := FALSE;
       "p15" := TRUE;
   END_IF;
   IF "t20" THEN
       "p15" := FALSE;
       "p16" := TRUE;
   END_IF;
   IF "t21" THEN
       "p16" := FALSE;
       "p17" := TRUE;
   END_IF;
   IF "t22" THEN
       "p17" := FALSE;
       "p23" := FALSE;
       "p24" := TRUE;
       "p22" := TRUE;
   END_IF;
   IF "t23" THEN
       "p18" := FALSE;
       "p19" := TRUE;
   END_IF;
   IF "t24" THEN
       "p19" := FALSE;
       "p2" := TRUE;
   END_IF;
   IF "t25" THEN
       "p17" := FALSE;
       "p22" := FALSE;
       "p25" := TRUE;
       "p23" := TRUE;
   END_IF;
   IF "t26" THEN
       "p20" := FALSE;
       "p21" := TRUE;
   END_IF;
   IF "t27" THEN
       "p21" := FALSE;
       "p27" := TRUE;
   END_IF;
   IF "t28" THEN
       "p24" := FALSE;
       "p18" := TRUE;
   END_IF;
   IF "t29" THEN
       "p25" := FALSE;
       "p20" := TRUE;
   END_IF;
   IF "t30" THEN
       "p21" := FALSE;
       "p26" := TRUE;
   END_IF;
   IF "t31" THEN
       "p26" := FALSE;
       "p2" := TRUE;
   END_IF;
   IF "t32" THEN
       "p27" := FALSE;
       "p2" := TRUE;
   END_IF;
END_REGION
END_FUNCTION

FUNCTION "Initialization" : Void   // FC3, LAD
{ S7_Optimized_Access := 'TRUE' }
VERSION : 0.1
BEGIN

REGION Network 1: Init
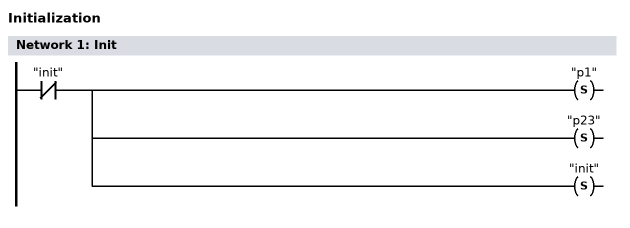
   RUNG wire#powerrail
      I_Contact( "init" )
      wire#w1
      S_Coil( "p1" )
   END_RUNG
   RUNG wire#w1
      S_Coil( "p23" )
   END_RUNG
   RUNG wire#w1
      S_Coil( "init" )
   END_RUNG
   // the same network as SCL:
   IF NOT "init" THEN
       "p1" := TRUE;
       "p23" := TRUE;
       "init" := TRUE;
   END_IF;
END_REGION
END_FUNCTION

FUNCTION "Actuators" : Void   // FC4, LAD
{ S7_Optimized_Access := 'TRUE' }
VERSION : 0.1
BEGIN

REGION Network 1: Actuators
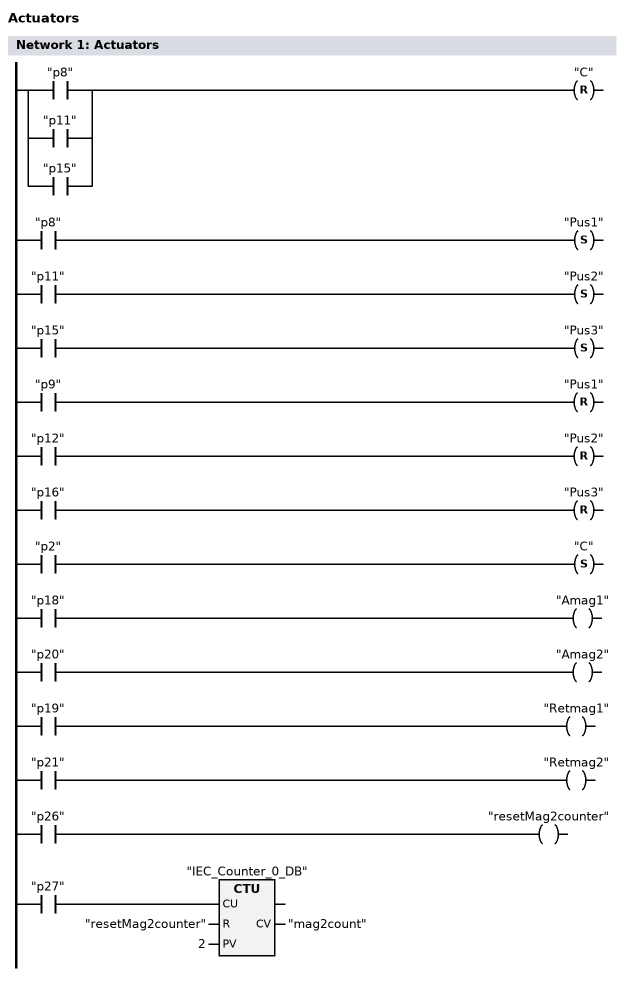
   IF "p8" OR "p11" OR "p15" THEN "C" := FALSE; END_IF;
   IF "p8" THEN "Pus1" := TRUE; END_IF;
   IF "p11" THEN "Pus2" := TRUE; END_IF;
   IF "p15" THEN "Pus3" := TRUE; END_IF;
   IF "p9" THEN "Pus1" := FALSE; END_IF;
   IF "p12" THEN "Pus2" := FALSE; END_IF;
   IF "p16" THEN "Pus3" := FALSE; END_IF;
   IF "p2" THEN "C" := TRUE; END_IF;
   "Amag1" := "p18";
   "Amag2" := "p20";
   "Retmag1" := "p19";
   "Retmag2" := "p21";
   "resetMag2counter" := "p26";
   "IEC_Counter_0_DB".CTU(CU := "p27", R := "resetMag2counter", PV := 2, CV => "mag2count");
END_REGION
END_FUNCTION

// ===== PLC "PLC_2"  Unspecific CPU 1500 =====

ORGANIZATION_BLOCK "Main"   // OB1, LAD, ProgramCycle
TITLE = "Main Program Sweep (Cycle)"
{ S7_Optimized_Access := 'TRUE' }
VERSION : 0.1
   VAR_INPUT
      Initial_Call : Bool;   // Initial call of this OB
      Remanence : Bool;   // =True, if remanent data are available
   END_VAR
BEGIN
END_ORGANIZATION_BLOCK